INTERFACE ITFLopendeBand

END_INTERFACE

(* stored: Version 1.1.0.1
   Itf ITFLopendeBand: Id {9d368c46-730b-40f0-8730-d7cbd8e44a65} *)
